FUNCTION_BLOCK Test_TEvent_AddEventHandler_ResizesListWhenListFull EXTENDS TUnitTestBase
VAR_INPUT
END_VAR
VAR_OUTPUT
END_VAR
VAR
    TestEvent : TTestEvent;
    TestEventHandler : TTestEventHandler;
END_VAR

TestEvent
    .ClearEventHandlers()
    .AddEventHandler(TestEventHandler)
    .AddEventHandler(TestEventHandler)
    .AddEventHandler(TestEventHandler)
    .AddEventHandler(TestEventHandler)
    .AddEventHandler(TestEventHandler)  // handler list now full - max handlers = 5
    .AddEventHandler(TestEventHandler); // should trigger an error message
    
Assertion.AssertEquals_UDINT(
    Expected := 6, // 
    Actual   := TestEvent.EventHandlers.Count,
    VariableName  := 'TestEvent.EventHandlers.Count');

TestFinished();

END_FUNCTION_BLOCK

(* stored: Version 1.1.0.1, ProductVersion 3.1.4024.4
   POU Test_TEvent_AddEventHandler_ResizesListWhenListFull: Id {88f9bb3e-8020-4cec-b239-7d266a547761}, SpecialFunc None *)
